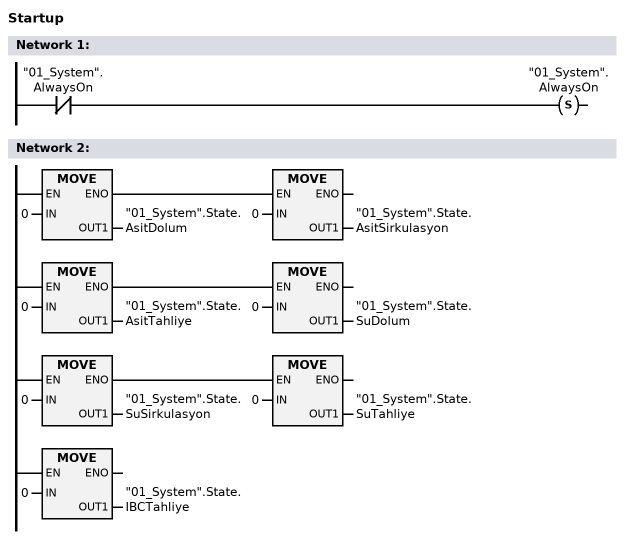
   RUNG wire#powerrail
      I_Contact( "01_System".AlwaysOn )
      S_Coil( "01_System".AlwaysOn )
   END_RUNG
   // the same network as SCL:
   IF NOT "01_System".AlwaysOn THEN "01_System".AlwaysOn := TRUE; END_IF;
END_REGION

REGION Network 2
   RUNG wire#powerrail
      Move(in := 0, out1 => "01_System".State.AsitDolum)
      Move(in := 0, out1 => "01_System".State.AsitSirkulasyon)
   END_RUNG
   RUNG wire#powerrail
      Move(in := 0, out1 => "01_System".State.AsitTahliye)
      Move(in := 0, out1 => "01_System".State.SuDolum)
   END_RUNG
   RUNG wire#powerrail
      Move(in := 0, out1 => "01_System".State.SuSirkulasyon)
      Move(in := 0, out1 => "01_System".State.SuTahliye)
   END_RUNG
   RUNG wire#powerrail
      Move(in := 0, out1 => "01_System".State.IBCTahliye)
   END_RUNG
   // the same network as SCL:
   "01_System".State.AsitDolum := 0;
   "01_System".State.AsitSirkulasyon := 0;
   "01_System".State.AsitTahliye := 0;
   "01_System".State.SuDolum := 0;
   "01_System".State.SuSirkulasyon := 0;
   "01_System".State.SuTahliye := 0;
   "01_System".State.IBCTahliye := 0;
END_REGION
END_ORGANIZATION_BLOCK